// TIA Portal V18 export
// export: Created 2026-06-08T16:32:20.618584Z, ExportSetting WithDefaults, DisplayName Totally Integrated Automation Portal, DisplayVersion V18, DisplayName TIA Portal Openness, DisplayVersion V18, DisplayName TIA Portal Version Control Interface, DisplayVersion V18, DisplayName STEP 7 Professional, DisplayVersion V18, DisplayName STEP 7 Safety, DisplayVersion V18, DisplayName WinCC Professional, DisplayVersion V18
DATA_BLOCK "LID_SORTING_STATION_DB"   // DB12
VERSION : 0.1
// stored: AutoNumber true, InstanceOfName LID_SORTING_STATION, InstanceOfType FB
"LID_SORTING_STATION"
BEGIN
END_DATA_BLOCK
